(* CoDeSys 2.3 export: WARNING_FB.EXP *)

(* POU FB/ФБ аварий/Warning_FB, ST *)
FUNCTION_BLOCK Warning_FB
VAR_INPUT
	input : BOOL;
END_VAR
VAR_OUTPUT
	bWarning: BOOL;
END_VAR
VAR
	TON1 : TON;
END_VAR
TON1(
	IN:=input ,
	PT:= T#5s  );

bWarning := SEL (TON1.Q, FALSE, TRUE );
END_FUNCTION_BLOCK
